Fanuc KAREL source: ko00079.KL

-- PROVISIONAL review KL for V1013-1; original PC SHA256 865835a12909ccdcb7f8c4c8995160122b19aa28f516e54de15e8f658f770610
-- Incomplete behavior may be omitted. Consult companion uncertainty JSON. Do not deploy.
PROGRAM KO00079
%NOLOCKGROUP
BEGIN
  -- UNRESOLVED_PC offsets 5-12; opcodes 9D,23
  -- UNRESOLVED_PC offsets 17-66; opcodes 27,22,1C,27,49,7E,AD,22,31,7E,4A
  -- UNRESOLVED_PC offsets 71-75; opcodes 7F
END KO00079
